// TIA Portal V20 export
TYPE "LKinCtrl_Diagnostics_typeHMIInterface"
// stored: Access Published
   STRUCT
      components : Word;
      layouts : Word;
      message : "LKinCtrl_Utilities_typeMessage";
      picker : "LKinCtrl_Picker_Kinematics_typeHMIInterface";
      overview : "LKinCtrl_OverviewDiagnostics_typeHMIInterface";
      technologyDiagnostics : Struct
         axis : "LKinCtrl_TechnologyDiagnostics_Axis_typeHMIInterface";
         kinematics : "LKinCtrl_TechnologyDiagnostics_Kinematics_typeHMIInterface";
      END_STRUCT;
   END_STRUCT;
END_TYPE
